// TIA Portal V20 export
// export: Created 2025-12-01T14:56:17.6270807Z, ExportSetting None, DisplayName Totally Integrated Automation Portal, DisplayVersion V20 Update 3, DisplayName TIA Portal Openness, DisplayVersion V20 Update 3, DisplayName TIA Portal Version Control Interface, DisplayVersion V20 Update 3, DisplayName STEP 7 Professional, DisplayVersion V20 Update 3, DisplayName STEP 7 Safety, DisplayVersion V20 Update 2, DisplayName WinCC Basic/Comfort/Advanced, DisplayVersion V20 Update 3, DisplayName WinCC Professional, DisplayVersion V20 Update 3, DisplayName WinCC Unified, DisplayVersion V20 Update 3
TYPE "UDT_ScadaDatosZona"
   STRUCT
      ErrorGrave : Bool;
      ErrorLeve : Bool;
      EmergenciaGrave : Bool;
      EmergenciaLeve : Bool;
      Libre_04 : Bool;
      FinReset : Bool;
      Memo_P_Marcha : Bool;
      Memo_P_Paro : Bool;
      MesasParo : Bool;
      MesasManual : Bool;
      MesasParoBlando : Bool;
      MesasError : Bool;
      MesasTodasEnParo : Bool;
      MesasTodasEnManual : Bool;
      Libre_16 : Bool;
      Libre_17 : Bool;
   END_STRUCT;
END_TYPE
